(* PLC project CoDeSys External Library Template, WAGO e!COCKPIT e!COCKPIT, author 3S - Smart Software Solutions GmbH *)
(* stored: creationDateTime 2019-10-29T12:37:19.6960561, version 3.5.5.30, modificationDateTime 2019-10-29T12:36:39.3744516, organization 3S - Smart Software Solutions GmbH *)
(* Library project template with all possible element types, docu and a sample project structure *)

FUNCTION_BLOCK fbPPPSLicznikCieplaMultical602
  VAR_INPUT
    sKomunikat : alSTRINGKomunikat;  (* komunikat z systemu zewnętrznego *)
    intTablicaKomunikatowRozmiar : INT;  (* rozmiar tablicy danych wysyłkowych *)
    intModbusOdczytZapisZadanieRozmiar : INT;  (* rozmiar tablicy danych modbusa *)
    xTablicaKomunikatowHold : BOOL;  (* wstrzymanie komunikacji mniej ważnych komunikatów *)
    sIdInstancji : STRING;  (* parametr ID rolety np NS02L*202IBM**** *)
    sIdAplikacji : STRING;  (* parametr ID aplikacji np SO*******ECL*000 *)
    sMnemonik : STRING;  (* mnemonik właściciela - BCB* *)
    sMACAdres : STRING;  (* MAC adres sterownika *)
    sDaneZapasowe : STRING;  (* 6 znaków zapasu *)
    tCzasOpoznieniaRestartu : TIME;  (* czas opóźnienia po którym zaczynają być raportowane wartości *)
    tCzasOpoznieniaAlarmu : TIME := TIME#1m0s0ms;  (* czas opóźnienia po którym zaczynają być raportowane wartości *)
    bAdres : BYTE;
    tMinimalnyCzasRaportowania : TIME;
    tMaksymalnyCzasRaportowania : TIME;
    xAutonomizacja : BOOL;
    xAutonomizacjaSztuczna : BOOL;
  END_VAR
  VAR_IN_OUT
    arModbusOdczytCykliczny : ARRAY[1..5000] OF typModbusOdczytCykliczny;
    arModbusStatusKomunikacji : ARRAY[1..256] OF INT;
    arTablicaKomunikatow : alARRAYTablicaKomunikatow;
    intTablicaKomunikatowZnacznikZapisu : INT;
  END_VAR
  VAR
    xPoInicjalizacji : BOOL := FALSE;  (* Inicjalizacja *)
    fbInicjalizacyjnyTimer : TON;
    tCzasInicjalizacji : TIME := TIME#30s0ms;
    xPierwszySkan : BOOL := TRUE;  (* Definicje zmiennych do odczytu wartości z modbusa *)
    intPetlaPierwszySkan : INT := 1;
    sDane : alSTRINGKomunikat;  (* Definicje do komunikacji z IZE *)
    sWyslanyKomunikat : alSTRINGKomunikat;
    sWyslanyKomunikatDummy : alSTRINGKomunikat;
    xZadanieRaportu : BOOL;
    sKomunikatPamiec : alSTRINGKomunikat;
    intPetla : INT;
    arErrorStan : ARRAY[0..10] OF INT;  (* tablica przechowująca statusy alarmowe *)
    arErrorKlasa : ARRAY[0..10] OF INT;  (* tablica przechowująca klasy danych alarmów *)
    xRaport : BOOL := FALSE;
    sTempWartoscAtrybutu : STRING;
    xOverFlow : BOOL;
    fbTimerBrakuKomunikacji : TON;  (* Kontrola komunikacji urządzenia *)
    xBrakKomunikacjiPLC : BOOL;
    xBrakKomunikacjiIZE : BOOL;
    wEnergiaCieplna_Lo : WORD;  (* Całkowita energia cieplna *)
    wEnergiaCieplna_Hi : WORD;
    rEnergiaCieplna : REAL;
    fbEnergiaCieplna : fbFiltrWartoscAnalogowa;
    rEnergiaCieplnaZaraportowana : REAL;
    wEnergiaCieplnaJednostka : WORD;  (* Jednostka energii cieplnej *)
    wPrzeplyw_Lo : WORD;  (* Aktualna wartość przepływu *)
    wPrzeplyw_Hi : WORD;
    rPrzeplyw : REAL;
    fbPrzeplyw : fbFiltrWartoscAnalogowa;
    rPrzeplywZaraportowana : REAL;
    wPrzeplywJednostka : REAL;  (* Jednostka przepływu *)
    rPrzeplywPamiec : REAL;  (* Wartosc przechowywana w pamieci w celu porównania z wartością aktualną *)
    xBrakZmianyPrzeplywu : BOOL;  (* Flaga informująca o braku zmiany przepływu w czasie *)
    fbBrakZmianyPrzeplywuTimer : TON;
    xBladBrakZmianyPrzeplywu : BOOL;  (* Flaga informująca o braku przeplywu przez czas 12h - podstawa wygenerowania alarmu *)
    wObjetosc_Lo : WORD;  (* Objętość medium, które przepłynęło przez licznik *)
    wObjetosc_Hi : WORD;
    rObjetosc : REAL;
    fbObjetosc : fbFiltrWartoscAnalogowa;
    rObjetoscZaraportowana : REAL;
    wObjetoscJednostka : WORD;  (* Jednostka wolumenu *)
    wMoc_Hi : WORD;  (* Aktualna moc cieplna płynąca przez licznik *)
    wMoc_Lo : WORD;
    rMoc : REAL;
    fbMoc : fbFiltrWartoscAnalogowa;
    rMocZaraportowana : REAL;
    wMocJednostka : WORD;  (* Jednostka mocy *)
    wTemperaturaZasilania_Lo : WORD;  (* Temp czynnika na wejściu licznika *)
    wTemperaturaZasilania_Hi : WORD;
    rTemperaturaZasilania : REAL;
    fbTemperaturaZasilania : fbFiltrWartoscAnalogowa;
    rTemperaturaZasilaniaZaraportowana : REAL;
    rTemperaturaZasilaniaPamiec : REAL;  (* Wartosc przechowywana w pamieci w celu porównania z wartością aktualną *)
    xBrakZmianyTemperaturyZasilania : BOOL;  (* Flaga informująca o braku zmiany przepływu w czasie *)
    fbBrakZmianyTemperaturyZasilaniaTimer : TON;
    xBladBrakZmianyTemperaturyZasilania : BOOL;  (* Flaga informująca o braku przeplywu przez czas 12h - podstawa wygenerowania alarmu *)
    wTemperaturaPowrotu_Lo : WORD;  (* Temp czynnika na wyjściu licznika *)
    wTemperaturaPowrotu_Hi : WORD;
    rTemperaturaPowrotu : REAL;
    fbTemperaturaPowrotu : fbFiltrWartoscAnalogowa;
    rTemperaturaPowrotuZaraportowana : REAL;
    rTemperaturaPowrotuPamiec : REAL;  (* Wartosc przechowywana w pamieci w celu porównania z wartością aktualną *)
    xBrakZmianyTemperaturyPowrotu : BOOL;  (* Flaga informująca o braku zmiany przepływu w czasie *)
    fbBrakZmianyTemperaturyPowrotuTimer : TON;
    xBladBrakZmianyTemperaturyPowrotu : BOOL;  (* Flaga informująca o braku przeplywu przez czas 12h - podstawa wygenerowania alarmu *)
  END_VAR

            (*			
Autor:					Jan Cichosz, 2019-03-25 
Prawa majątkowe: 		Solwena Sp. z o.o., 
Aktualizacje:			2019-05-16-AWy: Modyfikacja warunku na raportowanie. Dopisane: AND arModbusStatusKomunikacji[bAdres] = enumModbusStatus.KomunikacjaPrawidlowa AND xPoInicjalizacji
						2019-05-16-JC: Poprawki w formatowaniu, zmiany nazw zmiennych 
						2019-08-08-AWy: Zmiana nazw zmiennych i usunięcie zbędnych. Poprawki przy przeliczaniu zmiennych. Poprwaki w nazwach atrybutów. Generowanie alarmów czujników temperatury.
										Wysyłanie alarmów. Usunięcie blokady wykonywania rozkazów.
						2019-08-29-AWy: Zmiana poszczególnych parametrów przy przeliczaniu zmiennych. Usunięcie buga z raporotwania mocy.
					
Opis:					Komunikacja z licznikami ciepła Multical 602							
*)

// Inicjalizacja sterownika
fbInicjalizacyjnyTimer(IN := (NOT xPoInicjalizacji AND arModbusStatusKomunikacji[bAdres] = enumModbusStatus.KomunikacjaPrawidlowa), PT := tCzasOpoznieniaRestartu);
IF fbInicjalizacyjnyTimer.Q THEN
	rPrzeplywZaraportowana := rPrzeplyw;
	rMocZaraportowana := rMoc;
	rEnergiaCieplnaZaraportowana := rEnergiaCieplna;
	rObjetoscZaraportowana := rObjetosc;
	rTemperaturaZasilaniaZaraportowana := rTemperaturaZasilania;
	rTemperaturaPowrotuZaraportowana := rTemperaturaPowrotu;
	xPoInicjalizacji := TRUE;
END_IF

// Włącz autonomizację jeśli sterownik jest w stanie inicjalizacji lub nastąpiło wymuszenie autonomizacji
IF NOT xPoInicjalizacji OR xAutonomizacjaSztuczna = TRUE THEN
	xAutonomizacja := TRUE;
END_IF 

// Kontrola komunikacji
fbTimerBrakuKomunikacji(IN := arModbusStatusKomunikacji[bAdres] = enumModbusStatus.BrakKomunikacji, PT := T#60S);
IF fbTimerBrakuKomunikacji.Q THEN
	xBrakKomunikacjiPLC := TRUE;
ELSE
	xBrakKomunikacjiPLC := FALSE;
END_IF

IF xAutonomizacja THEN
	xBrakKomunikacjiIZE := TRUE;
ELSE
	xBrakKomunikacjiIZE := FALSE;
END_IF

// Deklaracja rejestrów Modbusa
IF xPierwszySkan THEN
	xPierwszySkan := FALSE;
	WHILE arModbusOdczytCykliczny[intPetlaPierwszySkan].bAdresUrzadzenia <> 0 DO
		intPetlaPierwszySkan := intPetlaPierwszySkan + 1;
	END_WHILE
	arModbusOdczytCykliczny[intPetlaPierwszySkan].bAdresUrzadzenia := bAdres;
	arModbusOdczytCykliczny[intPetlaPierwszySkan].bFunkcja := TO_BYTE(enumModbusKodyFunkcji.OdczytNRejestrow);
	arModbusOdczytCykliczny[intPetlaPierwszySkan].uiAdresRejestru := 256;
	arModbusOdczytCykliczny[intPetlaPierwszySkan].ltCzestotliwosc := TIME_TO_LTIME(tMinimalnyCzasRaportowania);
	arModbusOdczytCykliczny[intPetlaPierwszySkan].pZmiennaReferencyjna := ADR(wEnergiaCieplna_Hi);
	intPetlaPierwszySkan := intPetlaPierwszySkan + 1;	
	
	arModbusOdczytCykliczny[intPetlaPierwszySkan].bAdresUrzadzenia := bAdres;
	arModbusOdczytCykliczny[intPetlaPierwszySkan].bFunkcja := TO_BYTE(enumModbusKodyFunkcji.OdczytNRejestrow);
	arModbusOdczytCykliczny[intPetlaPierwszySkan].uiAdresRejestru := 257;
	arModbusOdczytCykliczny[intPetlaPierwszySkan].ltCzestotliwosc := TIME_TO_LTIME(tMinimalnyCzasRaportowania);
	arModbusOdczytCykliczny[intPetlaPierwszySkan].pZmiennaReferencyjna := ADR(wEnergiaCieplna_Lo);
	intPetlaPierwszySkan := intPetlaPierwszySkan + 1;
	
	arModbusOdczytCykliczny[intPetlaPierwszySkan].bAdresUrzadzenia := bAdres;
	arModbusOdczytCykliczny[intPetlaPierwszySkan].bFunkcja := TO_BYTE(enumModbusKodyFunkcji.OdczytNRejestrow);
	arModbusOdczytCykliczny[intPetlaPierwszySkan].uiAdresRejestru := 258;
	arModbusOdczytCykliczny[intPetlaPierwszySkan].ltCzestotliwosc := TIME_TO_LTIME(tMinimalnyCzasRaportowania);
	arModbusOdczytCykliczny[intPetlaPierwszySkan].pZmiennaReferencyjna := ADR(wPrzeplyw_Hi);
	intPetlaPierwszySkan := intPetlaPierwszySkan + 1;

	arModbusOdczytCykliczny[intPetlaPierwszySkan].bAdresUrzadzenia := bAdres;
	arModbusOdczytCykliczny[intPetlaPierwszySkan].bFunkcja := TO_BYTE(enumModbusKodyFunkcji.OdczytNRejestrow);
	arModbusOdczytCykliczny[intPetlaPierwszySkan].uiAdresRejestru := 259;
	arModbusOdczytCykliczny[intPetlaPierwszySkan].ltCzestotliwosc := TIME_TO_LTIME(tMinimalnyCzasRaportowania);
	arModbusOdczytCykliczny[intPetlaPierwszySkan].pZmiennaReferencyjna := ADR(wPrzeplyw_Lo);
	intPetlaPierwszySkan := intPetlaPierwszySkan + 1;
	
	arModbusOdczytCykliczny[intPetlaPierwszySkan].bAdresUrzadzenia := bAdres;
	arModbusOdczytCykliczny[intPetlaPierwszySkan].bFunkcja := TO_BYTE(enumModbusKodyFunkcji.OdczytNRejestrow);
	arModbusOdczytCykliczny[intPetlaPierwszySkan].uiAdresRejestru := 260;
	arModbusOdczytCykliczny[intPetlaPierwszySkan].ltCzestotliwosc := TIME_TO_LTIME(tMinimalnyCzasRaportowania);
	arModbusOdczytCykliczny[intPetlaPierwszySkan].pZmiennaReferencyjna := ADR(wObjetosc_Hi);
	intPetlaPierwszySkan := intPetlaPierwszySkan + 1;
	
	arModbusOdczytCykliczny[intPetlaPierwszySkan].bAdresUrzadzenia := bAdres;
	arModbusOdczytCykliczny[intPetlaPierwszySkan].bFunkcja := TO_BYTE(enumModbusKodyFunkcji.OdczytNRejestrow);
	arModbusOdczytCykliczny[intPetlaPierwszySkan].uiAdresRejestru := 261;
	arModbusOdczytCykliczny[intPetlaPierwszySkan].ltCzestotliwosc := TIME_TO_LTIME(tMinimalnyCzasRaportowania);
	arModbusOdczytCykliczny[intPetlaPierwszySkan].pZmiennaReferencyjna := ADR(wObjetosc_Lo);
	intPetlaPierwszySkan := intPetlaPierwszySkan + 1;
	
	arModbusOdczytCykliczny[intPetlaPierwszySkan].bAdresUrzadzenia := bAdres;
	arModbusOdczytCykliczny[intPetlaPierwszySkan].bFunkcja := TO_BYTE(enumModbusKodyFunkcji.OdczytNRejestrow);
	arModbusOdczytCykliczny[intPetlaPierwszySkan].uiAdresRejestru := 262;
	arModbusOdczytCykliczny[intPetlaPierwszySkan].ltCzestotliwosc := TIME_TO_LTIME(tMinimalnyCzasRaportowania);
	arModbusOdczytCykliczny[intPetlaPierwszySkan].pZmiennaReferencyjna := ADR(wMoc_Hi);
	intPetlaPierwszySkan := intPetlaPierwszySkan + 1;	
	
	arModbusOdczytCykliczny[intPetlaPierwszySkan].bAdresUrzadzenia := bAdres;
	arModbusOdczytCykliczny[intPetlaPierwszySkan].bFunkcja := TO_BYTE(enumModbusKodyFunkcji.OdczytNRejestrow);
	arModbusOdczytCykliczny[intPetlaPierwszySkan].uiAdresRejestru := 263;
	arModbusOdczytCykliczny[intPetlaPierwszySkan].ltCzestotliwosc := TIME_TO_LTIME(tMinimalnyCzasRaportowania);
	arModbusOdczytCykliczny[intPetlaPierwszySkan].pZmiennaReferencyjna := ADR(wMoc_Lo);
	intPetlaPierwszySkan := intPetlaPierwszySkan + 1;
	
	arModbusOdczytCykliczny[intPetlaPierwszySkan].bAdresUrzadzenia := bAdres;
	arModbusOdczytCykliczny[intPetlaPierwszySkan].bFunkcja := TO_BYTE(enumModbusKodyFunkcji.OdczytNRejestrow);
	arModbusOdczytCykliczny[intPetlaPierwszySkan].uiAdresRejestru := 264;
	arModbusOdczytCykliczny[intPetlaPierwszySkan].ltCzestotliwosc := TIME_TO_LTIME(tMinimalnyCzasRaportowania);
	arModbusOdczytCykliczny[intPetlaPierwszySkan].pZmiennaReferencyjna := ADR(wTemperaturaZasilania_Hi);
	intPetlaPierwszySkan := intPetlaPierwszySkan + 1;	
	
	arModbusOdczytCykliczny[intPetlaPierwszySkan].bAdresUrzadzenia := bAdres;
	arModbusOdczytCykliczny[intPetlaPierwszySkan].bFunkcja := TO_BYTE(enumModbusKodyFunkcji.OdczytNRejestrow);
	arModbusOdczytCykliczny[intPetlaPierwszySkan].uiAdresRejestru := 265;
	arModbusOdczytCykliczny[intPetlaPierwszySkan].ltCzestotliwosc := TIME_TO_LTIME(tMinimalnyCzasRaportowania);
	arModbusOdczytCykliczny[intPetlaPierwszySkan].pZmiennaReferencyjna := ADR(wTemperaturaZasilania_Lo);
	intPetlaPierwszySkan := intPetlaPierwszySkan + 1;
	
	arModbusOdczytCykliczny[intPetlaPierwszySkan].bAdresUrzadzenia := bAdres;
	arModbusOdczytCykliczny[intPetlaPierwszySkan].bFunkcja := TO_BYTE(enumModbusKodyFunkcji.OdczytNRejestrow);
	arModbusOdczytCykliczny[intPetlaPierwszySkan].uiAdresRejestru := 266;
	arModbusOdczytCykliczny[intPetlaPierwszySkan].ltCzestotliwosc := TIME_TO_LTIME(tMinimalnyCzasRaportowania);
	arModbusOdczytCykliczny[intPetlaPierwszySkan].pZmiennaReferencyjna := ADR(wTemperaturaPowrotu_Hi);
	intPetlaPierwszySkan := intPetlaPierwszySkan + 1;	
	
	arModbusOdczytCykliczny[intPetlaPierwszySkan].bAdresUrzadzenia := bAdres;
	arModbusOdczytCykliczny[intPetlaPierwszySkan].bFunkcja := TO_BYTE(enumModbusKodyFunkcji.OdczytNRejestrow);
	arModbusOdczytCykliczny[intPetlaPierwszySkan].uiAdresRejestru := 267;
	arModbusOdczytCykliczny[intPetlaPierwszySkan].ltCzestotliwosc := TIME_TO_LTIME(tMinimalnyCzasRaportowania);
	arModbusOdczytCykliczny[intPetlaPierwszySkan].pZmiennaReferencyjna := ADR(wTemperaturaPowrotu_Lo);
	intPetlaPierwszySkan := intPetlaPierwszySkan + 1;
		
	arModbusOdczytCykliczny[intPetlaPierwszySkan].bAdresUrzadzenia := bAdres;
	arModbusOdczytCykliczny[intPetlaPierwszySkan].bFunkcja := TO_BYTE(enumModbusKodyFunkcji.OdczytNRejestrow);
	arModbusOdczytCykliczny[intPetlaPierwszySkan].uiAdresRejestru := 272;
	arModbusOdczytCykliczny[intPetlaPierwszySkan].ltCzestotliwosc := TIME_TO_LTIME(tMinimalnyCzasRaportowania);
	arModbusOdczytCykliczny[intPetlaPierwszySkan].pZmiennaReferencyjna := ADR(wEnergiaCieplnaJednostka);
	intPetlaPierwszySkan := intPetlaPierwszySkan + 1;
	
	arModbusOdczytCykliczny[intPetlaPierwszySkan].bAdresUrzadzenia := bAdres;
	arModbusOdczytCykliczny[intPetlaPierwszySkan].bFunkcja := TO_BYTE(enumModbusKodyFunkcji.OdczytNRejestrow);
	arModbusOdczytCykliczny[intPetlaPierwszySkan].uiAdresRejestru := 273;
	arModbusOdczytCykliczny[intPetlaPierwszySkan].ltCzestotliwosc := TIME_TO_LTIME(tMinimalnyCzasRaportowania);
	arModbusOdczytCykliczny[intPetlaPierwszySkan].pZmiennaReferencyjna := ADR(wPrzeplywJednostka);
	intPetlaPierwszySkan := intPetlaPierwszySkan + 1;
	
	arModbusOdczytCykliczny[intPetlaPierwszySkan].bAdresUrzadzenia := bAdres;
	arModbusOdczytCykliczny[intPetlaPierwszySkan].bFunkcja := TO_BYTE(enumModbusKodyFunkcji.OdczytNRejestrow);
	arModbusOdczytCykliczny[intPetlaPierwszySkan].uiAdresRejestru := 274;
	arModbusOdczytCykliczny[intPetlaPierwszySkan].ltCzestotliwosc := TIME_TO_LTIME(tMinimalnyCzasRaportowania);
	arModbusOdczytCykliczny[intPetlaPierwszySkan].pZmiennaReferencyjna := ADR(wObjetoscJednostka);
	intPetlaPierwszySkan := intPetlaPierwszySkan + 1;
	
	arModbusOdczytCykliczny[intPetlaPierwszySkan].bAdresUrzadzenia := bAdres;
	arModbusOdczytCykliczny[intPetlaPierwszySkan].bFunkcja := TO_BYTE(enumModbusKodyFunkcji.OdczytNRejestrow);
	arModbusOdczytCykliczny[intPetlaPierwszySkan].uiAdresRejestru := 275;
	arModbusOdczytCykliczny[intPetlaPierwszySkan].ltCzestotliwosc := TIME_TO_LTIME(tMinimalnyCzasRaportowania);
	arModbusOdczytCykliczny[intPetlaPierwszySkan].pZmiennaReferencyjna := ADR(wMocJednostka);
	intPetlaPierwszySkan := intPetlaPierwszySkan + 1;
END_IF

// konwersja 2 odczytanych wordów na 32Float
fnKonwersja2x16naFloat32BySchneider(wRejestrMSW := wEnergiaCieplna_Hi, wRejestrLSW := wEnergiaCieplna_Lo, rWartoscFloat32 := rEnergiaCieplna);
fnKonwersja2x16naFloat32BySchneider(wRejestrMSW := wPrzeplyw_Hi, wRejestrLSW := wPrzeplyw_Lo, rWartoscFloat32 := rPrzeplyw);
fnKonwersja2x16naFloat32BySchneider(wRejestrMSW := wObjetosc_Hi, wRejestrLSW := wObjetosc_Lo, rWartoscFloat32 := rObjetosc);
fnKonwersja2x16naFloat32BySchneider(wRejestrMSW := wMoc_Hi, wRejestrLSW := wMoc_Lo, rWartoscFloat32 := rMoc);
fnKonwersja2x16naFloat32BySchneider(wRejestrMSW := wTemperaturaZasilania_Hi, wRejestrLSW := wTemperaturaZasilania_Lo, rWartoscFloat32 := rTemperaturaZasilania);
fnKonwersja2x16naFloat32BySchneider(wRejestrMSW := wTemperaturaPowrotu_Hi, wRejestrLSW := wTemperaturaPowrotu_Lo, rWartoscFloat32 := rTemperaturaPowrotu);

// Przeliczenie zmiennych
fbEnergiaCieplna(	rWartoscWejsciowa := rEnergiaCieplna,
					rDeadband := 100,
					tCzasMinimalny := tMinimalnyCzasRaportowania,
					tCzasMaksymalny := tMaksymalnyCzasRaportowania,
					rWynikMnoznik := 1000000000,
					rWynikOffset := 0,
					rWartoscWejsciowaZaraportowana := rEnergiaCieplnaZaraportowana,
					rWartoscWyjsciowa => rEnergiaCieplna);
					
fbPrzeplyw(	rWartoscWejsciowa := rPrzeplyw,
			rDeadband := 0.00000027778,
			tCzasMinimalny := tMinimalnyCzasRaportowania,
			tCzasMaksymalny := tMaksymalnyCzasRaportowania,
			rWynikMnoznik := 0.00000027778,
			rWynikOffset := 0,
			rWartoscWejsciowaZaraportowana := rPrzeplywZaraportowana,
			rWartoscWyjsciowa => rPrzeplyw);
							
fbObjetosc(	rWartoscWejsciowa := rObjetosc,
			rDeadband := 0.001,
			tCzasMinimalny := tMinimalnyCzasRaportowania,
			tCzasMaksymalny := tMaksymalnyCzasRaportowania,
			rWynikMnoznik := 1,
			rWynikOffset := 0,
			rWartoscWejsciowaZaraportowana := rObjetoscZaraportowana,
			rWartoscWyjsciowa => rObjetosc);								
								
fbMoc(	rWartoscWejsciowa := rMoc,
		rDeadband := 10,
		tCzasMinimalny := tMinimalnyCzasRaportowania,
		tCzasMaksymalny := tMaksymalnyCzasRaportowania,
		rWynikMnoznik := 1000,
		rWynikOffset := 0,
		rWartoscWejsciowaZaraportowana := rMocZaraportowana,
		rWartoscWyjsciowa => rMoc);
				
fbTemperaturaZasilania(	rWartoscWejsciowa := rTemperaturaZasilania,
						rDeadband := 0.1,
						tCzasMinimalny := tMinimalnyCzasRaportowania,
						tCzasMaksymalny := tMaksymalnyCzasRaportowania,
						rWynikMnoznik := 1,
						rWynikOffset := 273.15,
						rWartoscWejsciowaZaraportowana := rTemperaturaZasilaniaZaraportowana,
						rWartoscWyjsciowa => rTemperaturaZasilania);
			
fbTemperaturaPowrotu(	rWartoscWejsciowa := rTemperaturaPowrotu,
						rDeadband := 0.1,
						tCzasMinimalny := tMinimalnyCzasRaportowania,
						tCzasMaksymalny := tMaksymalnyCzasRaportowania,
						rWynikMnoznik := 1,
						rWynikOffset := 273.15,
						rWartoscWejsciowaZaraportowana := rTemperaturaPowrotuZaraportowana,
						rWartoscWyjsciowa => rTemperaturaPowrotu);							

// Sprawdzanie czy pomiar aktualnego przeplywu działa (alarm jest generowany, jeśli odczyt nie zmienił wartości w przeciągu 12h)
IF rPrzeplywPamiec = rPrzeplyw THEN
	xBrakZmianyPrzeplywu := TRUE;
ELSE
	xBrakZmianyPrzeplywu := FALSE;	
END_IF
fbBrakZmianyPrzeplywuTimer(IN := xBrakZmianyPrzeplywu, PT := T#12H);
IF fbBrakZmianyPrzeplywuTimer.Q THEN
	xBladBrakZmianyPrzeplywu := TRUE;
ELSE
	xBladBrakZmianyPrzeplywu := FALSE;
END_IF
rPrzeplywPamiec := rPrzeplyw;

// Sprawdzanie czy pomiar temperatury zasilania działa (alarm jest generowany, jeśli odczyt nie zmienił wartości w przeciągu 12h)
IF rTemperaturaZasilaniaPamiec = rTemperaturaZasilania THEN
	xBrakZmianyTemperaturyZasilania := TRUE;
ELSE
	xBrakZmianyTemperaturyZasilania := FALSE;	
END_IF
fbBrakZmianyTemperaturyZasilaniaTimer(IN := xBrakZmianyTemperaturyZasilania, PT := T#12H);
IF fbBrakZmianyTemperaturyZasilaniaTimer.Q THEN
	xBladBrakZmianyTemperaturyZasilania := TRUE;
ELSE
	xBladBrakZmianyTemperaturyZasilania := FALSE;
END_IF
rTemperaturaZasilaniaPamiec := rTemperaturaZasilania;

// Sprawdzanie czy pomiar temperatury powrotu działa (alarm jest generowany, jeśli odczyt nie zmienił wartości w przeciągu 12h)
IF rTemperaturaPowrotuPamiec = rTemperaturaPowrotu THEN
	xBrakZmianyTemperaturyPowrotu := TRUE;
ELSE
	xBrakZmianyTemperaturyPowrotu := FALSE;	
END_IF
fbBrakZmianyTemperaturyPowrotuTimer(IN := xBrakZmianyTemperaturyPowrotu, PT := T#12H);
IF fbBrakZmianyTemperaturyPowrotuTimer.Q THEN
	xBladBrakZmianyTemperaturyPowrotu := TRUE;
ELSE
	xBladBrakZmianyTemperaturyPowrotu := FALSE;
END_IF
rTemperaturaPowrotuPamiec := rTemperaturaPowrotu;

// Obsluga komunikatu przychodzacego z IZE
IF sKomunikat <> sKomunikatPamiec AND xPoInicjalizacji THEN
	sKomunikatPamiec := sKomunikat;
	IF fnIDOdbiorcyMatch(sKomunikat , sIdInstancji) THEN
		sDane := '';
		//zapytanie typu Q
		IF fnKomunikatTyp(sKomunikat) = 'Q' AND arModbusStatusKomunikacji[bAdres] = enumModbusStatus.KomunikacjaPrawidlowa THEN
			IF fnKomunikatDaneSzukajWartosci(sKomunikat , 'ENCC=') = '?' OR fnKomunikatDaneSzukajWartosci(sKomunikat , 'ALL=') = '?' THEN
				fnKomunikatDaneDodaj_xOverFlow(sDane := sDane , sAtrybut := 'ENCC=' , sWartosc := REAL_TO_STRING(rEnergiaCieplna) , xOverFlow := xOverFlow);	
				IF xOverFlow = TRUE THEN
					fnZapiszKomunikat(	sCalyKomunikat := '' ,
										sTypKomunikatu := 'A' ,
										sMnemonik := sMnemonik ,
										sMACAdres := sMACAdres ,
										sIDNadawcy := sIdInstancji ,
										sIDOdbiorcy := sIdAplikacji ,
										sDaneZapasowe := sDaneZapasowe ,
										sDane := sDane ,
										arTablicaKomunikatow := arTablicaKomunikatow ,
										intTablicaKomunikatowZnacznikZapisu := intTablicaKomunikatowZnacznikZapisu ,
										intTablicaKomunikatowRozmiar := intTablicaKomunikatowRozmiar ,
										sWyslanyKomunikat := sWyslanyKomunikatDummy);
					sDane := '';
				END_IF
			END_IF
			IF fnKomunikatDaneSzukajWartosci(sKomunikat , 'FLOWCC=') = '?' OR fnKomunikatDaneSzukajWartosci(sKomunikat , 'ALL=') = '?' THEN
				fnKomunikatDaneDodaj_xOverFlow(sDane := sDane , sAtrybut := 'FLOWCC=' , sWartosc := REAL_TO_STRING(rPrzeplyw) , xOverFlow := xOverFlow);	
				IF xOverFlow = TRUE THEN
					fnZapiszKomunikat(	sCalyKomunikat := '' ,
										sTypKomunikatu := 'A' ,
										sMnemonik := sMnemonik ,
										sMACAdres := sMACAdres ,
										sIDNadawcy := sIdInstancji ,
										sIDOdbiorcy := sIdAplikacji ,
										sDaneZapasowe := sDaneZapasowe ,
										sDane := sDane ,
										arTablicaKomunikatow := arTablicaKomunikatow ,
										intTablicaKomunikatowZnacznikZapisu := intTablicaKomunikatowZnacznikZapisu ,
										intTablicaKomunikatowRozmiar := intTablicaKomunikatowRozmiar ,
										sWyslanyKomunikat := sWyslanyKomunikatDummy);
					sDane := '';
				END_IF
			END_IF
			IF fnKomunikatDaneSzukajWartosci(sKomunikat , 'VOLCC=') = '?' OR fnKomunikatDaneSzukajWartosci(sKomunikat , 'ALL=') = '?' THEN
				fnKomunikatDaneDodaj_xOverFlow(sDane := sDane , sAtrybut := 'VOLCC=' , sWartosc := REAL_TO_STRING(rObjetosc) , xOverFlow := xOverFlow);	
				IF xOverFlow = TRUE THEN
					fnZapiszKomunikat(	sCalyKomunikat := '' ,
										sTypKomunikatu := 'A' ,
										sMnemonik := sMnemonik ,
										sMACAdres := sMACAdres ,
										sIDNadawcy := sIdInstancji ,
										sIDOdbiorcy := sIdAplikacji ,
										sDaneZapasowe := sDaneZapasowe ,
										sDane := sDane ,
										arTablicaKomunikatow := arTablicaKomunikatow ,
										intTablicaKomunikatowZnacznikZapisu := intTablicaKomunikatowZnacznikZapisu ,
										intTablicaKomunikatowRozmiar := intTablicaKomunikatowRozmiar ,
										sWyslanyKomunikat := sWyslanyKomunikatDummy);
					sDane := '';
				END_IF
			END_IF
			IF fnKomunikatDaneSzukajWartosci(sKomunikat , 'POWCC=') = '?' OR fnKomunikatDaneSzukajWartosci(sKomunikat , 'ALL=') = '?' THEN
				fnKomunikatDaneDodaj_xOverFlow(sDane := sDane , sAtrybut := 'POWCC=' , sWartosc := REAL_TO_STRING(rMoc) , xOverFlow := xOverFlow);	
				IF xOverFlow = TRUE THEN
					fnZapiszKomunikat(	sCalyKomunikat := '' ,
										sTypKomunikatu := 'A' ,
										sMnemonik := sMnemonik ,
										sMACAdres := sMACAdres ,
										sIDNadawcy := sIdInstancji ,
										sIDOdbiorcy := sIdAplikacji ,
										sDaneZapasowe := sDaneZapasowe ,
										sDane := sDane ,
										arTablicaKomunikatow := arTablicaKomunikatow ,
										intTablicaKomunikatowZnacznikZapisu := intTablicaKomunikatowZnacznikZapisu ,
										intTablicaKomunikatowRozmiar := intTablicaKomunikatowRozmiar ,
										sWyslanyKomunikat := sWyslanyKomunikatDummy);
					sDane := '';
				END_IF
			END_IF
			IF fnKomunikatDaneSzukajWartosci(sKomunikat , 'TEMPINCC=') = '?' OR fnKomunikatDaneSzukajWartosci(sKomunikat , 'ALL=') = '?' THEN
				fnKomunikatDaneDodaj_xOverFlow(sDane := sDane , sAtrybut := 'TEMPINCC=' , sWartosc := REAL_TO_STRING(rTemperaturaZasilania) , xOverFlow := xOverFlow);	
				IF xOverFlow = TRUE THEN
					fnZapiszKomunikat(	sCalyKomunikat := '' ,
										sTypKomunikatu := 'A' ,
										sMnemonik := sMnemonik ,
										sMACAdres := sMACAdres ,
										sIDNadawcy := sIdInstancji ,
										sIDOdbiorcy := sIdAplikacji ,
										sDaneZapasowe := sDaneZapasowe ,
										sDane := sDane ,
										arTablicaKomunikatow := arTablicaKomunikatow ,
										intTablicaKomunikatowZnacznikZapisu := intTablicaKomunikatowZnacznikZapisu ,
										intTablicaKomunikatowRozmiar := intTablicaKomunikatowRozmiar ,
										sWyslanyKomunikat := sWyslanyKomunikatDummy);
					sDane := '';
				END_IF
			END_IF
			IF fnKomunikatDaneSzukajWartosci(sKomunikat , 'TEMPOUTCC=') = '?' OR fnKomunikatDaneSzukajWartosci(sKomunikat , 'ALL=') = '?' THEN
				fnKomunikatDaneDodaj_xOverFlow(sDane := sDane , sAtrybut := 'TEMPOUTCC=' , sWartosc := REAL_TO_STRING(rTemperaturaPowrotu) , xOverFlow := xOverFlow);	
				IF xOverFlow = TRUE THEN
					fnZapiszKomunikat(	sCalyKomunikat := '' ,
										sTypKomunikatu := 'A' ,
										sMnemonik := sMnemonik ,
										sMACAdres := sMACAdres ,
										sIDNadawcy := sIdInstancji ,
										sIDOdbiorcy := sIdAplikacji ,
										sDaneZapasowe := sDaneZapasowe ,
										sDane := sDane ,
										arTablicaKomunikatow := arTablicaKomunikatow ,
										intTablicaKomunikatowZnacznikZapisu := intTablicaKomunikatowZnacznikZapisu ,
										intTablicaKomunikatowRozmiar := intTablicaKomunikatowRozmiar ,
										sWyslanyKomunikat := sWyslanyKomunikatDummy);
					sDane := '';
				END_IF
			END_IF
			// Pytanie o stany alarmów
			IF fnKomunikatDaneSzukajWartosci(sKomunikat , 'ALARM=') = '?' OR fnKomunikatDaneSzukajWartosci(sKomunikat , 'ALL=') = '?' THEN
				FOR intPetla := 1 TO 10 BY 1 DO
					// Raportowanie typu E (stanów alarmów) na zapytanie typu Q
					IF arErrorStan[intPetla] <> enumAlarmWartosc.StanNieznany THEN
						fnZapiszKomunikat(	sCalyKomunikat := '' ,
											sTypKomunikatu := 'E' ,
											sMnemonik := sMnemonik ,
											sMACAdres := sMACAdres ,
											sIDNadawcy := sIdInstancji ,
											sIDOdbiorcy := sIdAplikacji ,
											sDaneZapasowe := sDaneZapasowe ,
											sDane := fnKomunikatDaneErrorRetry(xAktywny := arErrorStan[intPetla] = enumAlarmWartosc.StanAlarmowy , intKlasa := arErrorKlasa[intPetla] , intNumer := intPetla),
											arTablicaKomunikatow := arTablicaKomunikatow ,
											intTablicaKomunikatowZnacznikZapisu := intTablicaKomunikatowZnacznikZapisu ,
											intTablicaKomunikatowRozmiar := intTablicaKomunikatowRozmiar ,
											sWyslanyKomunikat := sWyslanyKomunikatDummy);
					END_IF
				END_FOR
			END_IF
		END_IF
		// Raportowanie typu A na zapytanie Q
		IF sDane <> '' THEN
			fnZapiszKomunikat(	sCalyKomunikat := '' ,
								sTypKomunikatu := 'A' ,
								sMnemonik := sMnemonik ,
								sMACAdres := sMACAdres ,
								sIDNadawcy := sIdInstancji ,
								sIDOdbiorcy := sIdAplikacji ,
								sDaneZapasowe := sDaneZapasowe ,
								sDane := sDane ,
								arTablicaKomunikatow := arTablicaKomunikatow ,
								intTablicaKomunikatowZnacznikZapisu := intTablicaKomunikatowZnacznikZapisu ,
								intTablicaKomunikatowRozmiar := intTablicaKomunikatowRozmiar ,
								sWyslanyKomunikat := sWyslanyKomunikatDummy);
		END_IF
	END_IF
END_IF

// Raportowanie typu M do IZE wartosci odczytanych z Modbusa	
IF 	(rPrzeplyw <> rPrzeplywZaraportowana OR rMoc <> rMocZaraportowana OR rEnergiaCieplna <> rEnergiaCieplnaZaraportowana OR rObjetosc <> rObjetoscZaraportowana OR 
	rTemperaturaZasilania <> rTemperaturaZasilaniaZaraportowana OR rTemperaturaPowrotu <> rTemperaturaPowrotuZaraportowana) AND 
	arModbusStatusKomunikacji[bAdres] = enumModbusStatus.KomunikacjaPrawidlowa AND xPoInicjalizacji THEN
	xRaport := TRUE;
END_IF

IF xRaport THEN
	sDane := '';
	xRaport := FALSE;
	// Sumaryczna zużyta energia cieplna licznika
	IF rEnergiaCieplna <> rEnergiaCieplnaZaraportowana THEN
		rEnergiaCieplnaZaraportowana := rEnergiaCieplna;
		fnKomunikatDaneDodaj_xOverFlow(sDane := sDane , sAtrybut := 'ENCC=' , sWartosc := REAL_TO_STRING(rEnergiaCieplna) , xOverFlow := xOverFlow);	
		IF xOverFlow = TRUE THEN
			fnZapiszKomunikat(	sCalyKomunikat := '' ,
								sTypKomunikatu := 'M' ,
								sMnemonik := sMnemonik ,
								sMACAdres := sMACAdres ,
								sIDNadawcy := sIdInstancji ,
								sIDOdbiorcy := sIdAplikacji ,
								sDaneZapasowe := sDaneZapasowe ,
								sDane := sDane ,
								arTablicaKomunikatow := arTablicaKomunikatow ,
								intTablicaKomunikatowZnacznikZapisu := intTablicaKomunikatowZnacznikZapisu ,
								intTablicaKomunikatowRozmiar := intTablicaKomunikatowRozmiar ,
								sWyslanyKomunikat := sWyslanyKomunikatDummy);
			sDane := '';
		END_IF	
	END_IF
	// Biezacy przeplyw licznika 
	IF rPrzeplyw <> rPrzeplywZaraportowana THEN
		rPrzeplywZaraportowana := rPrzeplyw;
		fnKomunikatDaneDodaj_xOverFlow(sDane := sDane , sAtrybut := 'FLOWCC=' , sWartosc := REAL_TO_STRING(rPrzeplyw) , xOverFlow := xOverFlow);	
		IF xOverFlow = TRUE THEN
			fnZapiszKomunikat(	sCalyKomunikat := '' ,
								sTypKomunikatu := 'M' ,
								sMnemonik := sMnemonik ,
								sMACAdres := sMACAdres ,
								sIDNadawcy := sIdInstancji ,
								sIDOdbiorcy := sIdAplikacji ,
								sDaneZapasowe := sDaneZapasowe ,
								sDane := sDane ,
								arTablicaKomunikatow := arTablicaKomunikatow ,
								intTablicaKomunikatowZnacznikZapisu := intTablicaKomunikatowZnacznikZapisu ,
								intTablicaKomunikatowRozmiar := intTablicaKomunikatowRozmiar ,
								sWyslanyKomunikat := sWyslanyKomunikatDummy);
			sDane := '';
		END_IF	
	END_IF
	// Objętość medium, które przepłynęło przez licznik
	IF rObjetosc <> rObjetoscZaraportowana THEN
		rObjetoscZaraportowana := rObjetosc;
		fnKomunikatDaneDodaj_xOverFlow(sDane := sDane , sAtrybut := 'VOLCC=' , sWartosc := REAL_TO_STRING(rObjetosc) , xOverFlow := xOverFlow);	
		IF xOverFlow = TRUE THEN
			fnZapiszKomunikat(	sCalyKomunikat := '' ,
								sTypKomunikatu := 'M' ,
								sMnemonik := sMnemonik ,
								sMACAdres := sMACAdres ,
								sIDNadawcy := sIdInstancji ,
								sIDOdbiorcy := sIdAplikacji ,
								sDaneZapasowe := sDaneZapasowe ,
								sDane := sDane ,
								arTablicaKomunikatow := arTablicaKomunikatow ,
								intTablicaKomunikatowZnacznikZapisu := intTablicaKomunikatowZnacznikZapisu ,
								intTablicaKomunikatowRozmiar := intTablicaKomunikatowRozmiar ,
								sWyslanyKomunikat := sWyslanyKomunikatDummy);
			sDane := '';
		END_IF	
	END_IF
	// Biezaca moc licznika
	IF rMoc <> rMocZaraportowana THEN
		rMocZaraportowana := rMoc;
		fnKomunikatDaneDodaj_xOverFlow(sDane := sDane , sAtrybut := 'POWCC=' , sWartosc := REAL_TO_STRING(rMoc) , xOverFlow := xOverFlow);	
		IF xOverFlow = TRUE THEN
			fnZapiszKomunikat(	sCalyKomunikat := '' ,
								sTypKomunikatu := 'M' ,
								sMnemonik := sMnemonik ,
								sMACAdres := sMACAdres ,
								sIDNadawcy := sIdInstancji ,
								sIDOdbiorcy := sIdAplikacji ,
								sDaneZapasowe := sDaneZapasowe ,
								sDane := sDane ,
								arTablicaKomunikatow := arTablicaKomunikatow ,
								intTablicaKomunikatowZnacznikZapisu := intTablicaKomunikatowZnacznikZapisu ,
								intTablicaKomunikatowRozmiar := intTablicaKomunikatowRozmiar ,
								sWyslanyKomunikat := sWyslanyKomunikatDummy);
			sDane := '';
		END_IF	
	END_IF
	// Temperatura na wejsciu licznika
	IF rTemperaturaZasilania <> rTemperaturaZasilaniaZaraportowana THEN
		rTemperaturaZasilaniaZaraportowana := rTemperaturaZasilania;
		fnKomunikatDaneDodaj_xOverFlow(sDane := sDane , sAtrybut := 'TEMPINCC=' , sWartosc := REAL_TO_STRING(rTemperaturaZasilania) , xOverFlow := xOverFlow);	
		IF xOverFlow = TRUE THEN
			fnZapiszKomunikat(	sCalyKomunikat := '' ,
								sTypKomunikatu := 'M' ,
								sMnemonik := sMnemonik ,
								sMACAdres := sMACAdres ,
								sIDNadawcy := sIdInstancji ,
								sIDOdbiorcy := sIdAplikacji ,
								sDaneZapasowe := sDaneZapasowe ,
								sDane := sDane ,
								arTablicaKomunikatow := arTablicaKomunikatow ,
								intTablicaKomunikatowZnacznikZapisu := intTablicaKomunikatowZnacznikZapisu ,
								intTablicaKomunikatowRozmiar := intTablicaKomunikatowRozmiar ,
								sWyslanyKomunikat := sWyslanyKomunikatDummy);
			sDane := '';
		END_IF	
	END_IF
		// Temperatura na wyjsciu licznika
	IF rTemperaturaPowrotu <> rTemperaturaPowrotuZaraportowana THEN
		rTemperaturaPowrotuZaraportowana := rTemperaturaPowrotu;
		fnKomunikatDaneDodaj_xOverFlow(sDane := sDane , sAtrybut := 'TEMPOUTCC=' , sWartosc := REAL_TO_STRING(rTemperaturaPowrotu) , xOverFlow := xOverFlow);	
		IF xOverFlow = TRUE THEN
			fnZapiszKomunikat(	sCalyKomunikat := '' ,
								sTypKomunikatu := 'M' ,
								sMnemonik := sMnemonik ,
								sMACAdres := sMACAdres ,
								sIDNadawcy := sIdInstancji ,
								sIDOdbiorcy := sIdAplikacji ,
								sDaneZapasowe := sDaneZapasowe ,
								sDane := sDane ,
								arTablicaKomunikatow := arTablicaKomunikatow ,
								intTablicaKomunikatowZnacznikZapisu := intTablicaKomunikatowZnacznikZapisu ,
								intTablicaKomunikatowRozmiar := intTablicaKomunikatowRozmiar ,
								sWyslanyKomunikat := sWyslanyKomunikatDummy);
			sDane := '';
		END_IF	
	END_IF
	
	IF sDane <> '' AND xPoInicjalizacji THEN
		fnZapiszKomunikat(	sCalyKomunikat := '' ,
							sTypKomunikatu := 'M' ,
							sMnemonik := sMnemonik ,
							sMACAdres := sMACAdres ,
							sIDNadawcy := sIdInstancji ,
							sIDOdbiorcy := sIdAplikacji ,
							sDaneZapasowe := sDaneZapasowe ,
							sDane := sDane ,
							arTablicaKomunikatow := arTablicaKomunikatow ,
							intTablicaKomunikatowZnacznikZapisu := intTablicaKomunikatowZnacznikZapisu ,
							intTablicaKomunikatowRozmiar := intTablicaKomunikatowRozmiar ,
							sWyslanyKomunikat := sWyslanyKomunikat);
	END_IF
END_IF
	
// Alarm braku komunikacji MODBUS 
IF arErrorStan[enumPPPSLicznikCieplaMultical602Error.BrakKomunikacji] <> enumAlarmWartosc.StanAlarmowy AND arModbusStatusKomunikacji[bAdres] = enumModbusStatus.BrakKomunikacji THEN
	arErrorStan[enumPPPSLicznikCieplaMultical602Error.BrakKomunikacji] := enumAlarmWartosc.StanAlarmowy;
	arErrorKlasa[enumPPPSLicznikCieplaMultical602Error.BrakKomunikacji] := enumPPPSLicznikCieplaMultical602Error.BrakKomunikacji;
	IF xPoInicjalizacji THEN
		fnZapiszKomunikat(	sCalyKomunikat := '',
							sTypKomunikatu := 'E',
							sMnemonik := sMnemonik,
							sMACAdres := sMACAdres,
							sIDNadawcy := sIdInstancji,
							sIDOdbiorcy := sIdAplikacji,
							sDaneZapasowe := sDaneZapasowe,
							sDane := fnKomunikatDaneError(	xAktywny := TRUE, 
															intKlasa := enumPPPSLicznikCieplaMultical602ErrorKlasa.BrakKomunikacji, 
															intNumer := enumPPPSLicznikCieplaMultical602Error.BrakKomunikacji),
							arTablicaKomunikatow := arTablicaKomunikatow,
							intTablicaKomunikatowZnacznikZapisu := intTablicaKomunikatowZnacznikZapisu,
							intTablicaKomunikatowRozmiar := intTablicaKomunikatowRozmiar,
							sWyslanyKomunikat := sWyslanyKomunikatDummy);
	END_IF
END_IF
IF arErrorStan[enumPPPSLicznikCieplaMultical602Error.BrakKomunikacji] <> enumAlarmWartosc.StanNormalny AND arModbusStatusKomunikacji[bAdres] = enumModbusStatus.KomunikacjaPrawidlowa THEN
	arErrorStan[enumPPPSLicznikCieplaMultical602Error.BrakKomunikacji] := enumAlarmWartosc.StanNormalny;
	arErrorKlasa[enumPPPSLicznikCieplaMultical602Error.BrakKomunikacji] := enumPPPSLicznikCieplaMultical602Error.BrakKomunikacji;
	IF xPoInicjalizacji THEN
		fnZapiszKomunikat(	sCalyKomunikat := '',
							sTypKomunikatu := 'E',
							sMnemonik := sMnemonik,
							sMACAdres := sMACAdres,
							sIDNadawcy := sIdInstancji,
							sIDOdbiorcy := sIdAplikacji,
							sDaneZapasowe := sDaneZapasowe,
							sDane := fnKomunikatDaneError(	xAktywny := FALSE, 
															intKlasa := enumPPPSLicznikCieplaMultical602ErrorKlasa.BrakKomunikacji, 
															intNumer := enumPPPSLicznikCieplaMultical602Error.BrakKomunikacji),
							arTablicaKomunikatow := arTablicaKomunikatow,
							intTablicaKomunikatowZnacznikZapisu := intTablicaKomunikatowZnacznikZapisu,
							intTablicaKomunikatowRozmiar := intTablicaKomunikatowRozmiar,
							sWyslanyKomunikat := sWyslanyKomunikatDummy);
	END_IF
END_IF
	
// Alarm czujnika przepływu
IF arErrorStan[enumPPPSLicznikCieplaMultical602Error.AlarmCzujnikaPrzeplywu] <> enumAlarmWartosc.StanAlarmowy AND xBladBrakZmianyPrzeplywu THEN
	arErrorStan[enumPPPSLicznikCieplaMultical602Error.AlarmCzujnikaPrzeplywu] := enumAlarmWartosc.StanAlarmowy;
	arErrorKlasa[enumPPPSLicznikCieplaMultical602Error.AlarmCzujnikaPrzeplywu] := enumPPPSLicznikCieplaMultical602Error.AlarmCzujnikaPrzeplywu;
	IF xPoInicjalizacji THEN
		fnZapiszKomunikat(	sCalyKomunikat := '',
							sTypKomunikatu := 'E',
							sMnemonik := sMnemonik,
							sMACAdres := sMACAdres,
							sIDNadawcy := sIdInstancji,
							sIDOdbiorcy := sIdAplikacji,
							sDaneZapasowe := sDaneZapasowe,
							sDane := fnKomunikatDaneError(	xAktywny := TRUE, 
															intKlasa := enumPPPSLicznikCieplaMultical602ErrorKlasa.AlarmCzujnikaPrzeplywu, 
															intNumer := enumPPPSLicznikCieplaMultical602Error.AlarmCzujnikaPrzeplywu),
							arTablicaKomunikatow := arTablicaKomunikatow,
							intTablicaKomunikatowZnacznikZapisu := intTablicaKomunikatowZnacznikZapisu,
							intTablicaKomunikatowRozmiar := intTablicaKomunikatowRozmiar,
							sWyslanyKomunikat := sWyslanyKomunikatDummy);
	END_IF
END_IF
IF arErrorStan[enumPPPSLicznikCieplaMultical602Error.AlarmCzujnikaPrzeplywu] <> enumAlarmWartosc.StanNormalny AND NOT xBladBrakZmianyPrzeplywu THEN
	arErrorStan[enumPPPSLicznikCieplaMultical602Error.AlarmCzujnikaPrzeplywu] := enumAlarmWartosc.StanNormalny;
	arErrorKlasa[enumPPPSLicznikCieplaMultical602Error.AlarmCzujnikaPrzeplywu] := enumPPPSLicznikCieplaMultical602Error.AlarmCzujnikaPrzeplywu;
	IF xPoInicjalizacji THEN
		fnZapiszKomunikat(	sCalyKomunikat := '',
							sTypKomunikatu := 'E',
							sMnemonik := sMnemonik,
							sMACAdres := sMACAdres,
							sIDNadawcy := sIdInstancji,
							sIDOdbiorcy := sIdAplikacji,
							sDaneZapasowe := sDaneZapasowe,
							sDane := fnKomunikatDaneError(	xAktywny := FALSE, 
															intKlasa := enumPPPSLicznikCieplaMultical602ErrorKlasa.AlarmCzujnikaPrzeplywu, 
															intNumer := enumPPPSLicznikCieplaMultical602Error.AlarmCzujnikaPrzeplywu),
							arTablicaKomunikatow := arTablicaKomunikatow,
							intTablicaKomunikatowZnacznikZapisu := intTablicaKomunikatowZnacznikZapisu,
							intTablicaKomunikatowRozmiar := intTablicaKomunikatowRozmiar ,
							sWyslanyKomunikat := sWyslanyKomunikatDummy);
	END_IF
END_IF
	
// Alarm czujnika temperatury zasilania
IF arErrorStan[enumPPPSLicznikCieplaMultical602Error.AlarmCzujnikaZasilania] <> enumAlarmWartosc.StanAlarmowy AND xBladBrakZmianyTemperaturyZasilania THEN
	arErrorStan[enumPPPSLicznikCieplaMultical602Error.AlarmCzujnikaZasilania] := enumAlarmWartosc.StanAlarmowy;
	arErrorKlasa[enumPPPSLicznikCieplaMultical602Error.AlarmCzujnikaZasilania] := enumPPPSLicznikCieplaMultical602Error.AlarmCzujnikaZasilania;
	IF xPoInicjalizacji THEN
		fnZapiszKomunikat(	sCalyKomunikat := '',
							sTypKomunikatu := 'E',
							sMnemonik := sMnemonik,
							sMACAdres := sMACAdres,
							sIDNadawcy := sIdInstancji,
							sIDOdbiorcy := sIdAplikacji,
							sDaneZapasowe := sDaneZapasowe,
							sDane := fnKomunikatDaneError(	xAktywny := TRUE, 
														  	intKlasa := enumPPPSLicznikCieplaMultical602ErrorKlasa.AlarmCzujnikaZasilania, 
															intNumer := enumPPPSLicznikCieplaMultical602Error.AlarmCzujnikaZasilania),
							arTablicaKomunikatow := arTablicaKomunikatow,
							intTablicaKomunikatowZnacznikZapisu := intTablicaKomunikatowZnacznikZapisu,
							intTablicaKomunikatowRozmiar := intTablicaKomunikatowRozmiar,
							sWyslanyKomunikat := sWyslanyKomunikatDummy);
	END_IF
END_IF
IF arErrorStan[enumPPPSLicznikCieplaMultical602Error.AlarmCzujnikaZasilania] <> enumAlarmWartosc.StanNormalny AND NOT xBladBrakZmianyTemperaturyZasilania THEN
	arErrorStan[enumPPPSLicznikCieplaMultical602Error.AlarmCzujnikaZasilania] := enumAlarmWartosc.StanNormalny;
	arErrorKlasa[enumPPPSLicznikCieplaMultical602Error.AlarmCzujnikaZasilania] := enumPPPSLicznikCieplaMultical602Error.AlarmCzujnikaZasilania;
	IF xPoInicjalizacji THEN
		fnZapiszKomunikat(	sCalyKomunikat := '',
							sTypKomunikatu := 'E',
							sMnemonik := sMnemonik,
							sMACAdres := sMACAdres,
							sIDNadawcy := sIdInstancji,
							sIDOdbiorcy := sIdAplikacji,
							sDaneZapasowe := sDaneZapasowe,
							sDane := fnKomunikatDaneError(	xAktywny := FALSE, 
															intKlasa := enumPPPSLicznikCieplaMultical602ErrorKlasa.AlarmCzujnikaZasilania, 
															intNumer := enumPPPSLicznikCieplaMultical602Error.AlarmCzujnikaZasilania),
							arTablicaKomunikatow := arTablicaKomunikatow,
							intTablicaKomunikatowZnacznikZapisu := intTablicaKomunikatowZnacznikZapisu,
							intTablicaKomunikatowRozmiar := intTablicaKomunikatowRozmiar ,
							sWyslanyKomunikat := sWyslanyKomunikatDummy);
	END_IF
END_IF	
	
// Alarm czujnika temperatury powrotu
IF arErrorStan[enumPPPSLicznikCieplaMultical602Error.AlarmCzujnikaPowrotu] <> enumAlarmWartosc.StanAlarmowy AND xBladBrakZmianyTemperaturyPowrotu THEN
	arErrorStan[enumPPPSLicznikCieplaMultical602Error.AlarmCzujnikaPowrotu] := enumAlarmWartosc.StanAlarmowy;
	arErrorKlasa[enumPPPSLicznikCieplaMultical602Error.AlarmCzujnikaPowrotu] := enumPPPSLicznikCieplaMultical602Error.AlarmCzujnikaPowrotu;
	IF xPoInicjalizacji THEN
		fnZapiszKomunikat(	sCalyKomunikat := '',
							sTypKomunikatu := 'E',
							sMnemonik := sMnemonik,
							sMACAdres := sMACAdres,
							sIDNadawcy := sIdInstancji,
							sIDOdbiorcy := sIdAplikacji,
							sDaneZapasowe := sDaneZapasowe,
							sDane := fnKomunikatDaneError(	xAktywny := TRUE, 
															intKlasa := enumPPPSLicznikCieplaMultical602ErrorKlasa.AlarmCzujnikaPowrotu, 
															intNumer := enumPPPSLicznikCieplaMultical602Error.AlarmCzujnikaPowrotu),
							arTablicaKomunikatow := arTablicaKomunikatow,
							intTablicaKomunikatowZnacznikZapisu := intTablicaKomunikatowZnacznikZapisu,
							intTablicaKomunikatowRozmiar := intTablicaKomunikatowRozmiar,
							sWyslanyKomunikat := sWyslanyKomunikatDummy);
	END_IF
END_IF
IF arErrorStan[enumPPPSLicznikCieplaMultical602Error.AlarmCzujnikaPowrotu] <> enumAlarmWartosc.StanNormalny AND NOT xBladBrakZmianyTemperaturyPowrotu THEN
	arErrorStan[enumPPPSLicznikCieplaMultical602Error.AlarmCzujnikaPowrotu] := enumAlarmWartosc.StanNormalny;
	arErrorKlasa[enumPPPSLicznikCieplaMultical602Error.AlarmCzujnikaPowrotu] := enumPPPSLicznikCieplaMultical602Error.AlarmCzujnikaPowrotu;
	IF xPoInicjalizacji THEN
		fnZapiszKomunikat(	sCalyKomunikat := '',
							sTypKomunikatu := 'E',
							sMnemonik := sMnemonik,
							sMACAdres := sMACAdres,
							sIDNadawcy := sIdInstancji,
							sIDOdbiorcy := sIdAplikacji,
							sDaneZapasowe := sDaneZapasowe,
							sDane := fnKomunikatDaneError(	xAktywny := FALSE, 
															intKlasa := enumPPPSLicznikCieplaMultical602ErrorKlasa.AlarmCzujnikaPowrotu, 
															intNumer := enumPPPSLicznikCieplaMultical602Error.AlarmCzujnikaPowrotu),
							arTablicaKomunikatow := arTablicaKomunikatow,
							intTablicaKomunikatowZnacznikZapisu := intTablicaKomunikatowZnacznikZapisu,
							intTablicaKomunikatowRozmiar := intTablicaKomunikatowRozmiar ,
							sWyslanyKomunikat := sWyslanyKomunikatDummy);
	END_IF
END_IF

          
END_FUNCTION_BLOCK
